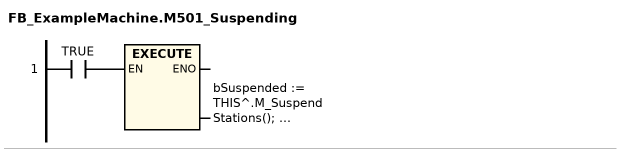
// NETWORK 1
bSuspended := THIS^.M_SuspendStations();
END_METHOD

(* In this state the most recent execution status should be maintained while
awaiting an explicit 'Unsuspend' command once external conditions are satisfactory. *)
METHOD M511_Suspended : BOOL
VAR_OUTPUT
	(* This should be set to true if an explicit 'Unsuspend' command is received.
	Once set to true, the state machine will move to the 'Unsuspending' state. *)
	bUnsuspend	: BOOL;
	(* This should be set to true if an external source requests that the module
	exit its current state and come to a controlled stop. Once set to true, the
	state machine will move to the 'Stopping' state. *)
	bStop	: BOOL;
	(* This should be set to true if a potentially hazardous error or a safety
	fault has occurred in any tasks. Once set to true, the state machine will
	move to the 'Aborting' state. *)
	bAbort	: BOOL;
END_VAR
// NETWORK 1
END_METHOD

(* In this state, the module and its components should be returned to the
scenario it was in before it entered the 'Suspending' step so that the
'Execute' state can pick up where it left off. *)
METHOD M521_Unsuspending : BOOL
VAR_OUTPUT
	(* This should be set to true once the module is ready to restart
	execution. Once set to true, the state machine will move to the 'Execute'
	state. *)
	bUnsuspended	: BOOL;
	(* This should be set to true if an external source requests that the module
	exit its current state and come to a controlled stop. Once set to true, the
	state machine will move to the 'Stopping' state. *)
	bStop	: BOOL;
	(* This should be set to true if a potentially hazardous error or a safety
	fault has occurred in any tasks. Once set to true, the state machine will
	move to the 'Aborting' state. *)
	bAbort	: BOOL;
END_VAR
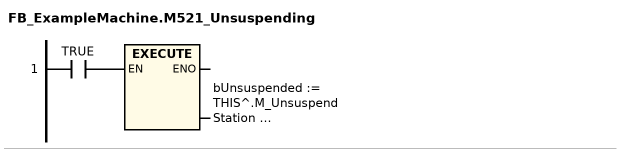
// NETWORK 1
bUnsuspended := THIS^.M_UnsuspendStations();
END_METHOD

END_FUNCTION_BLOCK

// ---- 1 Module/1 Stations/FB_ExampleStation.TcPOU
FUNCTION_BLOCK FB_ExampleStation EXTENDS FB_Station
VAR_INPUT
	in_fbDevice : REFERENCE TO FB_Device;
END_VAR
VAR_OUTPUT
END_VAR
VAR
END_VAR

THIS^.A_StateMachine();

END_FUNCTION_BLOCK

// ---- 1 Module/2 Devices/FB_ExampleDevice.TcPOU
FUNCTION_BLOCK FB_ExampleDevice EXTENDS FB_Device
VAR_INPUT
END_VAR
VAR_OUTPUT
END_VAR
VAR
END_VAR

END_FUNCTION_BLOCK
